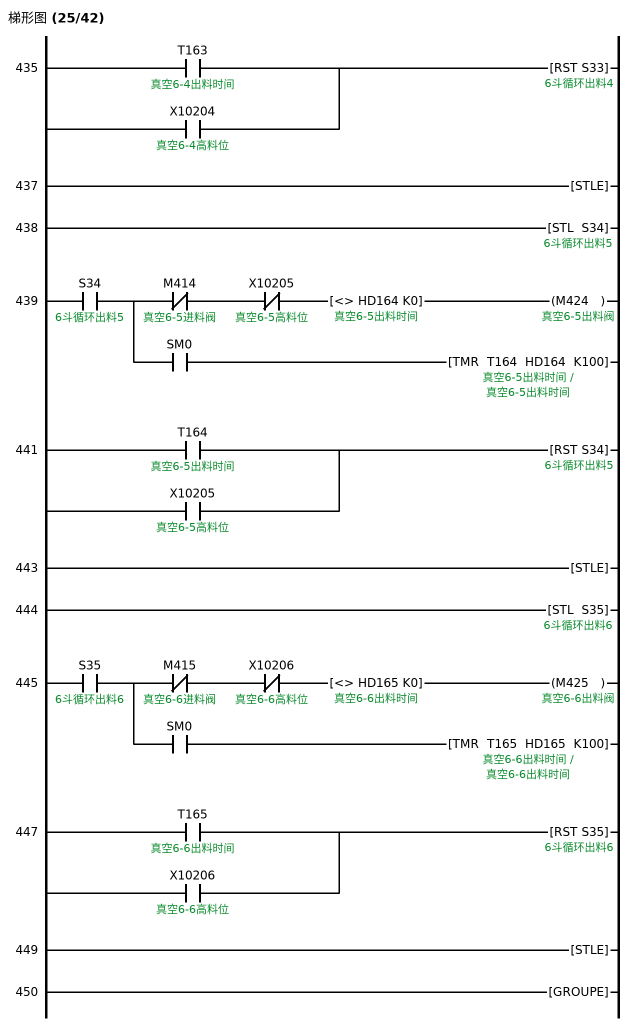
[picture p24: 梯形图 rows 435-450]
LD     T163	; 真空6-4出料时间
OR     X10204	; 真空6-4高料位
RST    S33	; 6斗循环出料4
STLE
STL    S34	; 6斗循环出料5
LD     S34	; 6斗循环出料5
MPS
ANI    M414	; 真空6-5进料阀
ANI    X10205	; 真空6-5高料位
AND<>  HD164 K0	; 真空6-5出料时间
OUT    M424	; 真空6-5出料阀
MPP
AND    SM0
TMR    T164 HD164 K100	; 真空6-5出料时间 / 真空6-5出料时间
LD     T164	; 真空6-5出料时间
OR     X10205	; 真空6-5高料位
RST    S34	; 6斗循环出料5
STLE
STL    S35	; 6斗循环出料6
LD     S35	; 6斗循环出料6
MPS
ANI    M415	; 真空6-6进料阀
ANI    X10206	; 真空6-6高料位
AND<>  HD165 K0	; 真空6-6出料时间
OUT    M425	; 真空6-6出料阀
MPP
AND    SM0
TMR    T165 HD165 K100	; 真空6-6出料时间 / 真空6-6出料时间
LD     T165	; 真空6-6出料时间
OR     X10206	; 真空6-6高料位
RST    S35	; 6斗循环出料6
STLE
GROUPE

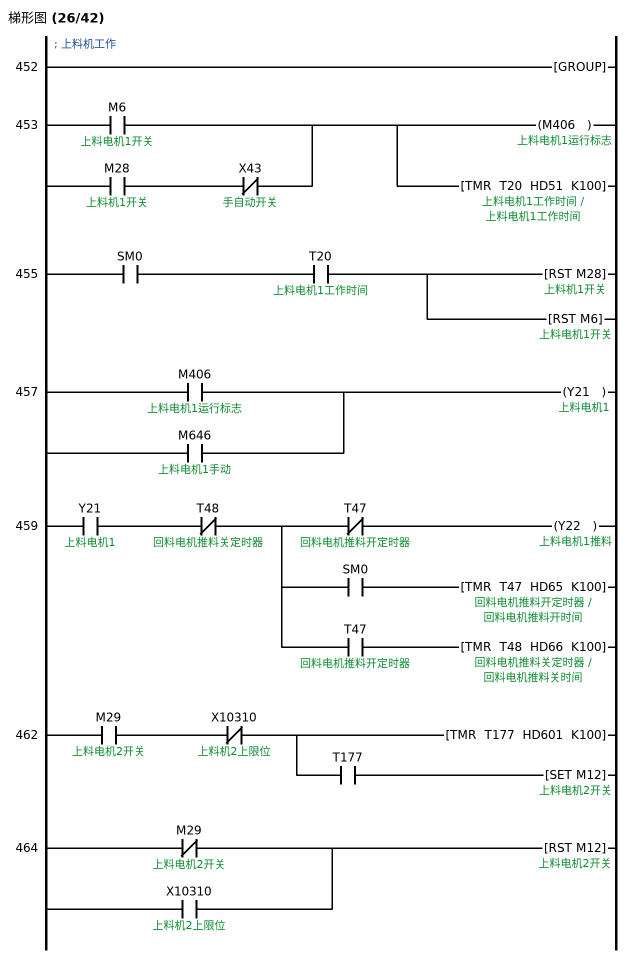
; 上料机工作
GROUP
LD     M6	; 上料电机1开关
LD     M28	; 上料机1开关
ANI    X43	; 手自动开关
ORB
OUT    M406	; 上料电机1运行标志
TMR    T20 HD51 K100	; 上料电机1工作时间 / 上料电机1工作时间
LD     SM0
AND    T20	; 上料电机1工作时间
RST    M28	; 上料机1开关
RST    M6	; 上料电机1开关
LD     M406	; 上料电机1运行标志
OR     M646	; 上料电机1手动
OUT    Y21	; 上料电机1
LD     Y21	; 上料电机1
ANI    T48	; 回料电机推料关定时器
MPS
ANI    T47	; 回料电机推料开定时器
OUT    Y22	; 上料电机1推料
MRD
AND    SM0
TMR    T47 HD65 K100	; 回料电机推料开定时器 / 回料电机推料开时间
MPP
AND    T47	; 回料电机推料开定时器
TMR    T48 HD66 K100	; 回料电机推料关定时器 / 回料电机推料关时间
LD     M29	; 上料电机2开关
ANI    X10310	; 上料机2上限位
TMR    T177 HD601 K100
AND    T177
SET    M12	; 上料电机2开关
LDI    M29	; 上料电机2开关
OR     X10310	; 上料机2上限位
RST    M12	; 上料电机2开关

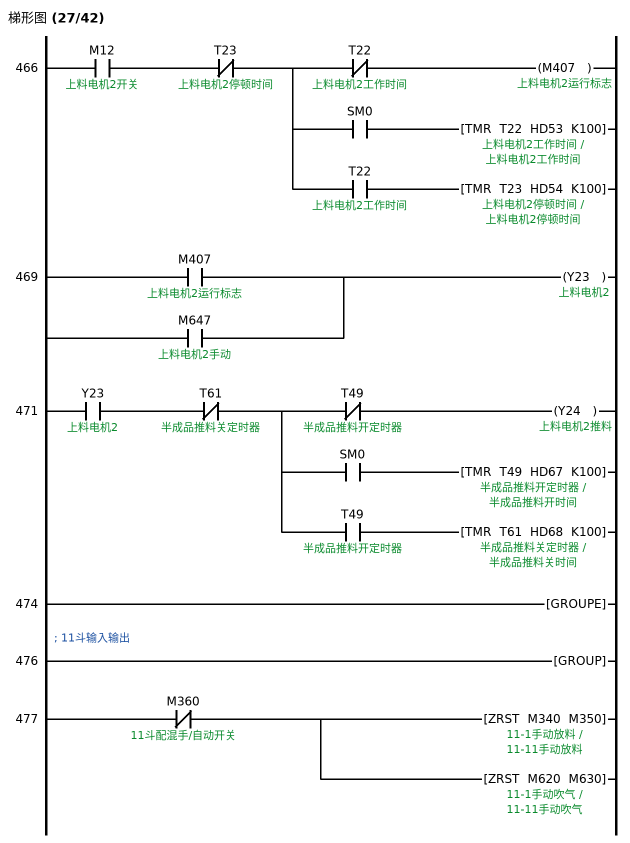
LD     M12	; 上料电机2开关
ANI    T23	; 上料电机2停顿时间
MPS
ANI    T22	; 上料电机2工作时间
OUT    M407	; 上料电机2运行标志
MRD
AND    SM0
TMR    T22 HD53 K100	; 上料电机2工作时间 / 上料电机2工作时间
MPP
AND    T22	; 上料电机2工作时间
TMR    T23 HD54 K100	; 上料电机2停顿时间 / 上料电机2停顿时间
LD     M407	; 上料电机2运行标志
OR     M647	; 上料电机2手动
OUT    Y23	; 上料电机2
LD     Y23	; 上料电机2
ANI    T61	; 半成品推料关定时器
MPS
ANI    T49	; 半成品推料开定时器
OUT    Y24	; 上料电机2推料
MRD
AND    SM0
TMR    T49 HD67 K100	; 半成品推料开定时器 / 半成品推料开时间
MPP
AND    T49	; 半成品推料开定时器
TMR    T61 HD68 K100	; 半成品推料关定时器 / 半成品推料关时间
GROUPE
; 11斗输入输出
GROUP
LDI    M360	; 11斗配混手/自动开关
ZRST   M340 M350	; 11-1手动放料 / 11-11手动放料
ZRST   M620 M630	; 11-1手动吹气 / 11-11手动吹气

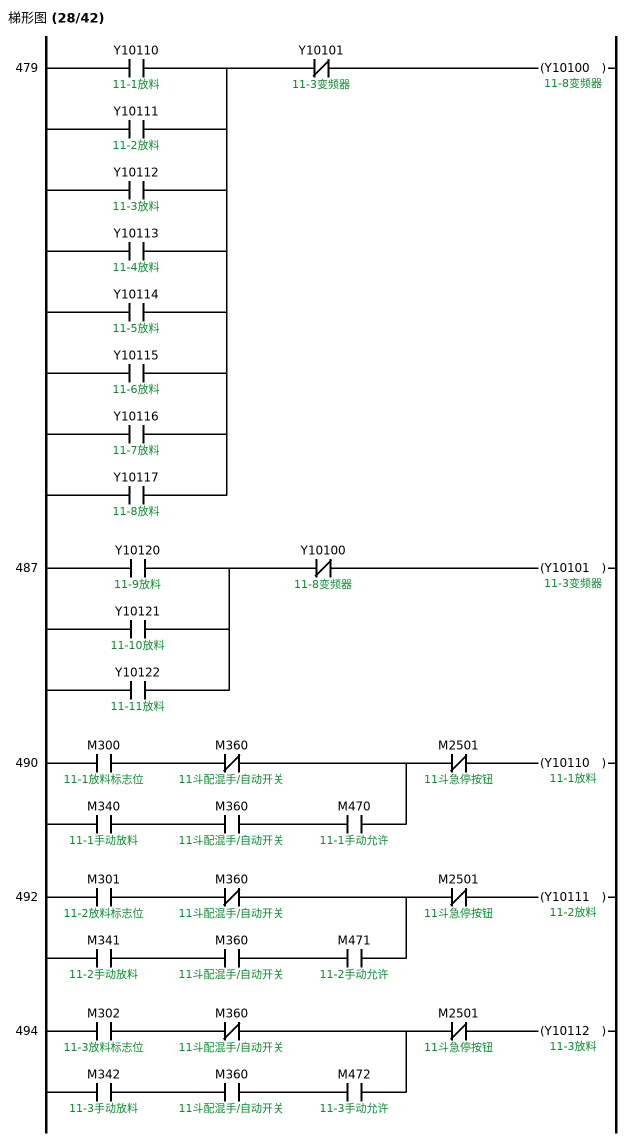
LD     Y10110	; 11-1放料
OR     Y10111	; 11-2放料
OR     Y10112	; 11-3放料
OR     Y10113	; 11-4放料
OR     Y10114	; 11-5放料
OR     Y10115	; 11-6放料
OR     Y10116	; 11-7放料
OR     Y10117	; 11-8放料
ANI    Y10101	; 11-3变频器
OUT    Y10100	; 11-8变频器
LD     Y10120	; 11-9放料
OR     Y10121	; 11-10放料
OR     Y10122	; 11-11放料
ANI    Y10100	; 11-8变频器
OUT    Y10101	; 11-3变频器
LD     M300	; 11-1放料标志位
ANI    M360	; 11斗配混手/自动开关
LD     M340	; 11-1手动放料
AND    M360	; 11斗配混手/自动开关
AND    M470	; 11-1手动允许
ORB
ANI    M2501	; 11斗急停按钮
OUT    Y10110	; 11-1放料
LD     M301	; 11-2放料标志位
ANI    M360	; 11斗配混手/自动开关
LD     M341	; 11-2手动放料
AND    M360	; 11斗配混手/自动开关
AND    M471	; 11-2手动允许
ORB
ANI    M2501	; 11斗急停按钮
OUT    Y10111	; 11-2放料
LD     M302	; 11-3放料标志位
ANI    M360	; 11斗配混手/自动开关
LD     M342	; 11-3手动放料
AND    M360	; 11斗配混手/自动开关
AND    M472	; 11-3手动允许
ORB
ANI    M2501	; 11斗急停按钮
OUT    Y10112	; 11-3放料

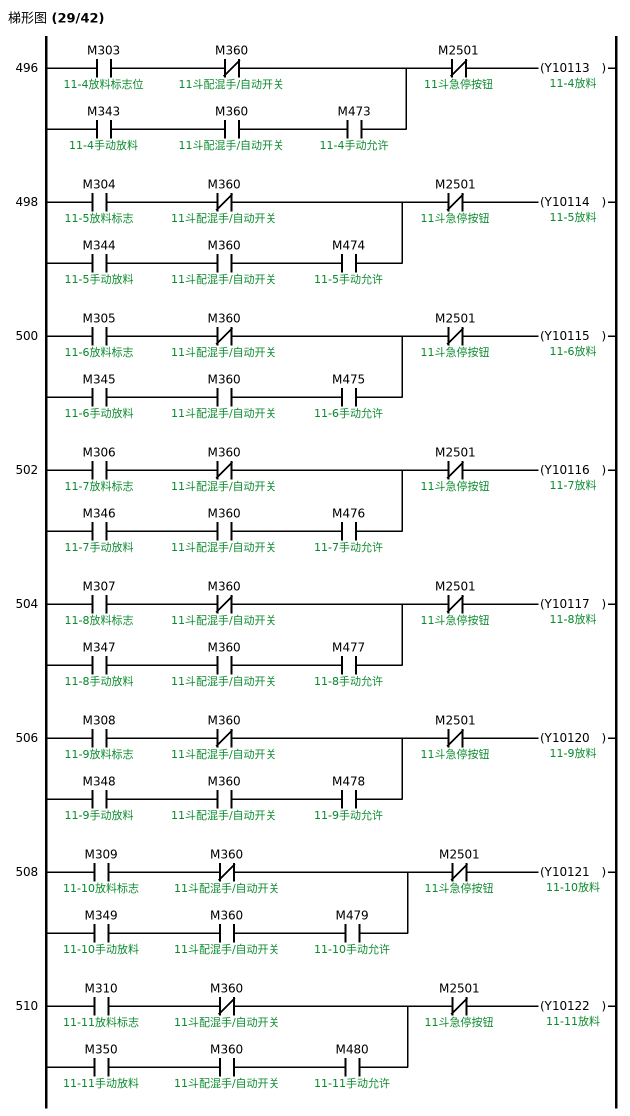
LD     M303	; 11-4放料标志位
ANI    M360	; 11斗配混手/自动开关
LD     M343	; 11-4手动放料
AND    M360	; 11斗配混手/自动开关
AND    M473	; 11-4手动允许
ORB
ANI    M2501	; 11斗急停按钮
OUT    Y10113	; 11-4放料
LD     M304	; 11-5放料标志
ANI    M360	; 11斗配混手/自动开关
LD     M344	; 11-5手动放料
AND    M360	; 11斗配混手/自动开关
AND    M474	; 11-5手动允许
ORB
ANI    M2501	; 11斗急停按钮
OUT    Y10114	; 11-5放料
LD     M305	; 11-6放料标志
ANI    M360	; 11斗配混手/自动开关
LD     M345	; 11-6手动放料
AND    M360	; 11斗配混手/自动开关
AND    M475	; 11-6手动允许
ORB
ANI    M2501	; 11斗急停按钮
OUT    Y10115	; 11-6放料
LD     M306	; 11-7放料标志
ANI    M360	; 11斗配混手/自动开关
LD     M346	; 11-7手动放料
AND    M360	; 11斗配混手/自动开关
AND    M476	; 11-7手动允许
ORB
ANI    M2501	; 11斗急停按钮
OUT    Y10116	; 11-7放料
LD     M307	; 11-8放料标志
ANI    M360	; 11斗配混手/自动开关
LD     M347	; 11-8手动放料
AND    M360	; 11斗配混手/自动开关
AND    M477	; 11-8手动允许
ORB
ANI    M2501	; 11斗急停按钮
OUT    Y10117	; 11-8放料
LD     M308	; 11-9放料标志
ANI    M360	; 11斗配混手/自动开关
LD     M348	; 11-9手动放料
AND    M360	; 11斗配混手/自动开关
AND    M478	; 11-9手动允许
ORB
ANI    M2501	; 11斗急停按钮
OUT    Y10120	; 11-9放料
LD     M309	; 11-10放料标志
ANI    M360	; 11斗配混手/自动开关
LD     M349	; 11-10手动放料
AND    M360	; 11斗配混手/自动开关
AND    M479	; 11-10手动允许
ORB
ANI    M2501	; 11斗急停按钮
OUT    Y10121	; 11-10放料
LD     M310	; 11-11放料标志
ANI    M360	; 11斗配混手/自动开关
LD     M350	; 11-11手动放料
AND    M360	; 11斗配混手/自动开关
AND    M480	; 11-11手动允许
ORB
ANI    M2501	; 11斗急停按钮
OUT    Y10122	; 11-11放料

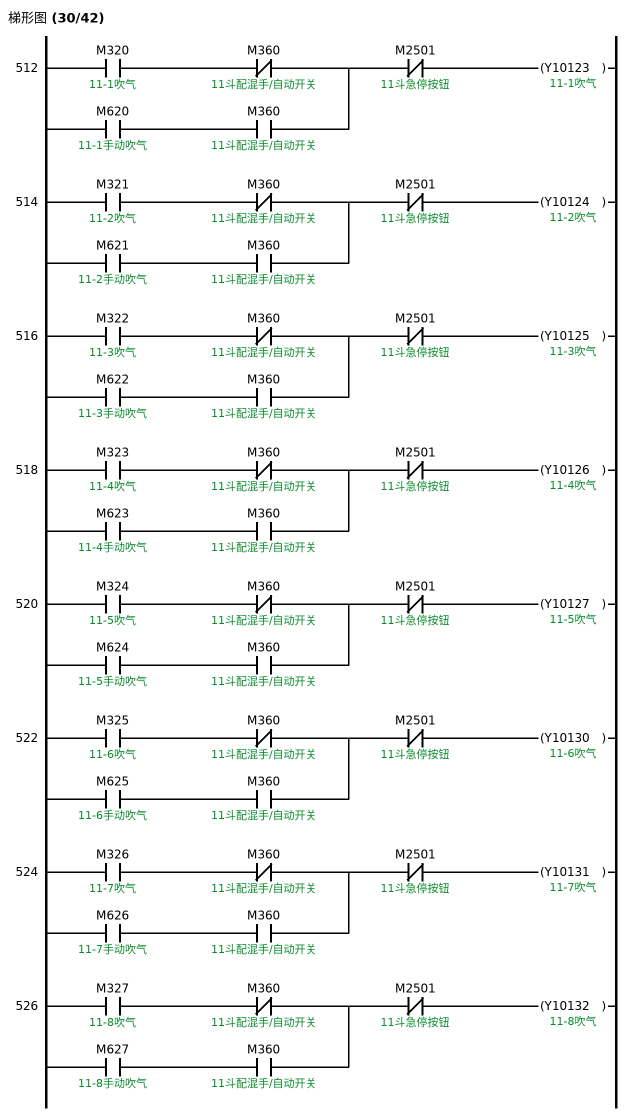
LD     M320	; 11-1吹气
ANI    M360	; 11斗配混手/自动开关
LD     M620	; 11-1手动吹气
AND    M360	; 11斗配混手/自动开关
ORB
ANI    M2501	; 11斗急停按钮
OUT    Y10123	; 11-1吹气
LD     M321	; 11-2吹气
ANI    M360	; 11斗配混手/自动开关
LD     M621	; 11-2手动吹气
AND    M360	; 11斗配混手/自动开关
ORB
ANI    M2501	; 11斗急停按钮
OUT    Y10124	; 11-2吹气
LD     M322	; 11-3吹气
ANI    M360	; 11斗配混手/自动开关
LD     M622	; 11-3手动吹气
AND    M360	; 11斗配混手/自动开关
ORB
ANI    M2501	; 11斗急停按钮
OUT    Y10125	; 11-3吹气
LD     M323	; 11-4吹气
ANI    M360	; 11斗配混手/自动开关
LD     M623	; 11-4手动吹气
AND    M360	; 11斗配混手/自动开关
ORB
ANI    M2501	; 11斗急停按钮
OUT    Y10126	; 11-4吹气
LD     M324	; 11-5吹气
ANI    M360	; 11斗配混手/自动开关
LD     M624	; 11-5手动吹气
AND    M360	; 11斗配混手/自动开关
ORB
ANI    M2501	; 11斗急停按钮
OUT    Y10127	; 11-5吹气
LD     M325	; 11-6吹气
ANI    M360	; 11斗配混手/自动开关
LD     M625	; 11-6手动吹气
AND    M360	; 11斗配混手/自动开关
ORB
ANI    M2501	; 11斗急停按钮
OUT    Y10130	; 11-6吹气
LD     M326	; 11-7吹气
ANI    M360	; 11斗配混手/自动开关
LD     M626	; 11-7手动吹气
AND    M360	; 11斗配混手/自动开关
ORB
ANI    M2501	; 11斗急停按钮
OUT    Y10131	; 11-7吹气
LD     M327	; 11-8吹气
ANI    M360	; 11斗配混手/自动开关
LD     M627	; 11-8手动吹气
AND    M360	; 11斗配混手/自动开关
ORB
ANI    M2501	; 11斗急停按钮
OUT    Y10132	; 11-8吹气

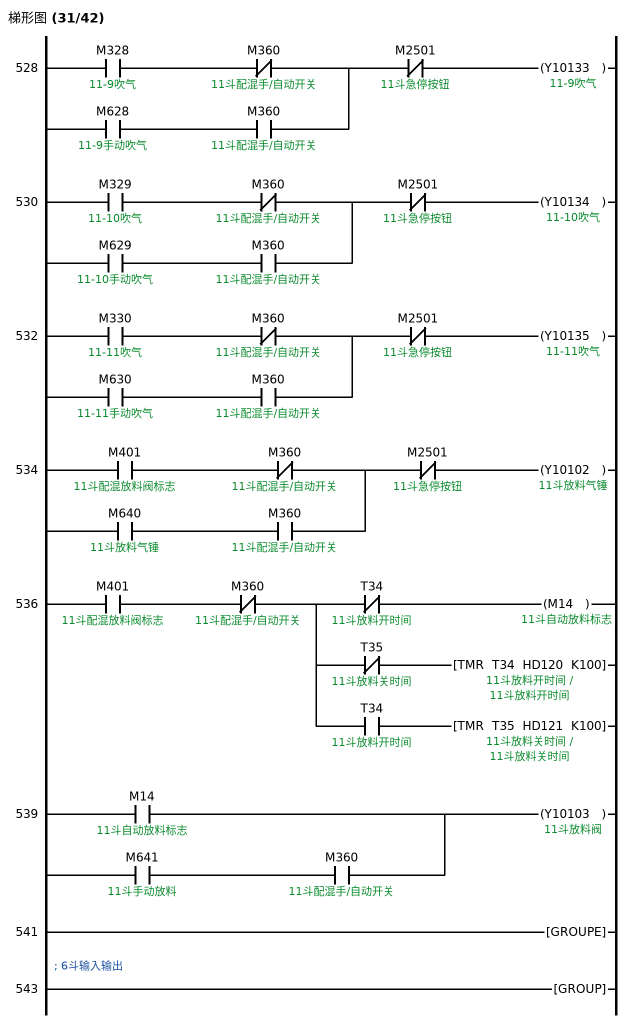
LD     M328	; 11-9吹气
ANI    M360	; 11斗配混手/自动开关
LD     M628	; 11-9手动吹气
AND    M360	; 11斗配混手/自动开关
ORB
ANI    M2501	; 11斗急停按钮
OUT    Y10133	; 11-9吹气
LD     M329	; 11-10吹气
ANI    M360	; 11斗配混手/自动开关
LD     M629	; 11-10手动吹气
AND    M360	; 11斗配混手/自动开关
ORB
ANI    M2501	; 11斗急停按钮
OUT    Y10134	; 11-10吹气
LD     M330	; 11-11吹气
ANI    M360	; 11斗配混手/自动开关
LD     M630	; 11-11手动吹气
AND    M360	; 11斗配混手/自动开关
ORB
ANI    M2501	; 11斗急停按钮
OUT    Y10135	; 11-11吹气
LD     M401	; 11斗配混放料阀标志
ANI    M360	; 11斗配混手/自动开关
LD     M640	; 11斗放料气锤
AND    M360	; 11斗配混手/自动开关
ORB
ANI    M2501	; 11斗急停按钮
OUT    Y10102	; 11斗放料气锤
LD     M401	; 11斗配混放料阀标志
ANI    M360	; 11斗配混手/自动开关
MPS
ANI    T34	; 11斗放料开时间
OUT    M14	; 11斗自动放料标志
MRD
ANI    T35	; 11斗放料关时间
TMR    T34 HD120 K100	; 11斗放料开时间 / 11斗放料开时间
MPP
AND    T34	; 11斗放料开时间
TMR    T35 HD121 K100	; 11斗放料关时间 / 11斗放料关时间
LD     M14	; 11斗自动放料标志
LD     M641	; 11斗手动放料
AND    M360	; 11斗配混手/自动开关
ORB
OUT    Y10103	; 11斗放料阀
GROUPE
; 6斗输入输出
GROUP

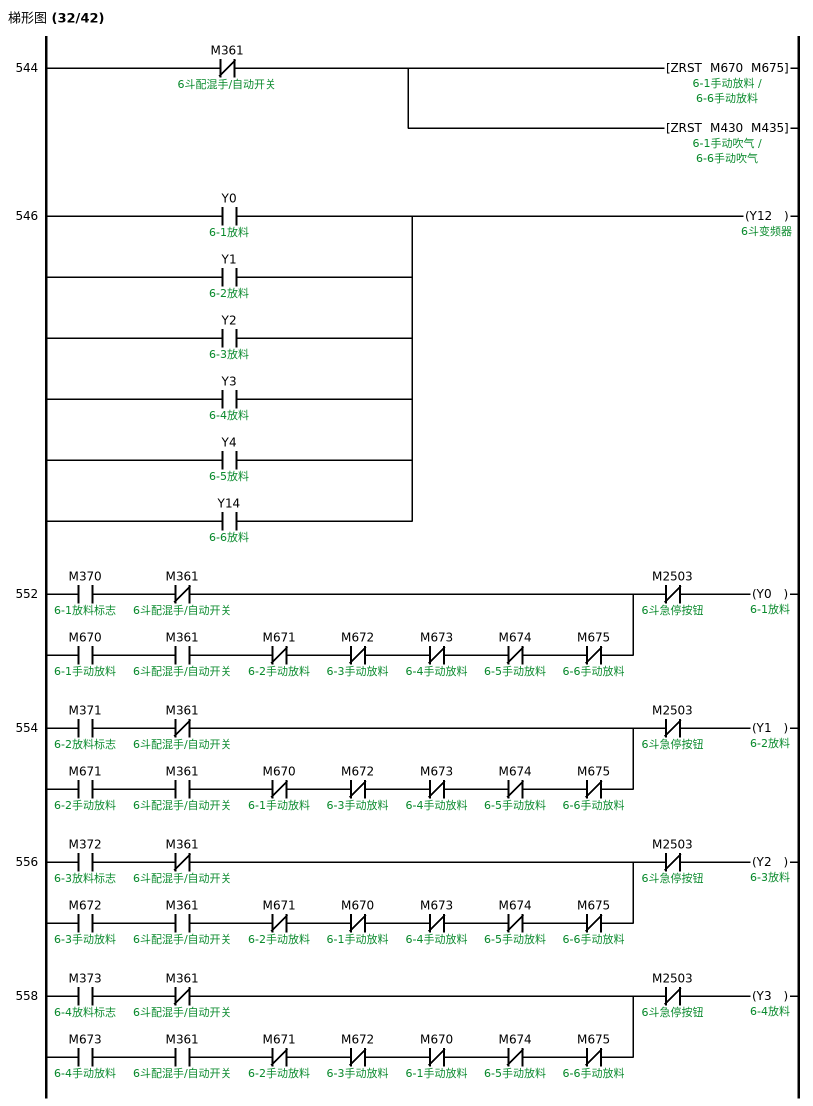
LDI    M361	; 6斗配混手/自动开关
ZRST   M670 M675	; 6-1手动放料 / 6-6手动放料
ZRST   M430 M435	; 6-1手动吹气 / 6-6手动吹气
LD     Y0	; 6-1放料
OR     Y1	; 6-2放料
OR     Y2	; 6-3放料
OR     Y3	; 6-4放料
OR     Y4	; 6-5放料
OR     Y14	; 6-6放料
OUT    Y12	; 6斗变频器
LD     M370	; 6-1放料标志
ANI    M361	; 6斗配混手/自动开关
LD     M670	; 6-1手动放料
AND    M361	; 6斗配混手/自动开关
ANI    M671	; 6-2手动放料
ANI    M672	; 6-3手动放料
ANI    M673	; 6-4手动放料
ANI    M674	; 6-5手动放料
ANI    M675	; 6-6手动放料
ORB
ANI    M2503	; 6斗急停按钮
OUT    Y0	; 6-1放料
LD     M371	; 6-2放料标志
ANI    M361	; 6斗配混手/自动开关
LD     M671	; 6-2手动放料
AND    M361	; 6斗配混手/自动开关
ANI    M670	; 6-1手动放料
ANI    M672	; 6-3手动放料
ANI    M673	; 6-4手动放料
ANI    M674	; 6-5手动放料
ANI    M675	; 6-6手动放料
ORB
ANI    M2503	; 6斗急停按钮
OUT    Y1	; 6-2放料
LD     M372	; 6-3放料标志
ANI    M361	; 6斗配混手/自动开关
LD     M672	; 6-3手动放料
AND    M361	; 6斗配混手/自动开关
ANI    M671	; 6-2手动放料
ANI    M670	; 6-1手动放料
ANI    M673	; 6-4手动放料
ANI    M674	; 6-5手动放料
ANI    M675	; 6-6手动放料
ORB
ANI    M2503	; 6斗急停按钮
OUT    Y2	; 6-3放料
LD     M373	; 6-4放料标志
ANI    M361	; 6斗配混手/自动开关
LD     M673	; 6-4手动放料
AND    M361	; 6斗配混手/自动开关
ANI    M671	; 6-2手动放料
ANI    M672	; 6-3手动放料
ANI    M670	; 6-1手动放料
ANI    M674	; 6-5手动放料
ANI    M675	; 6-6手动放料
ORB
ANI    M2503	; 6斗急停按钮
OUT    Y3	; 6-4放料

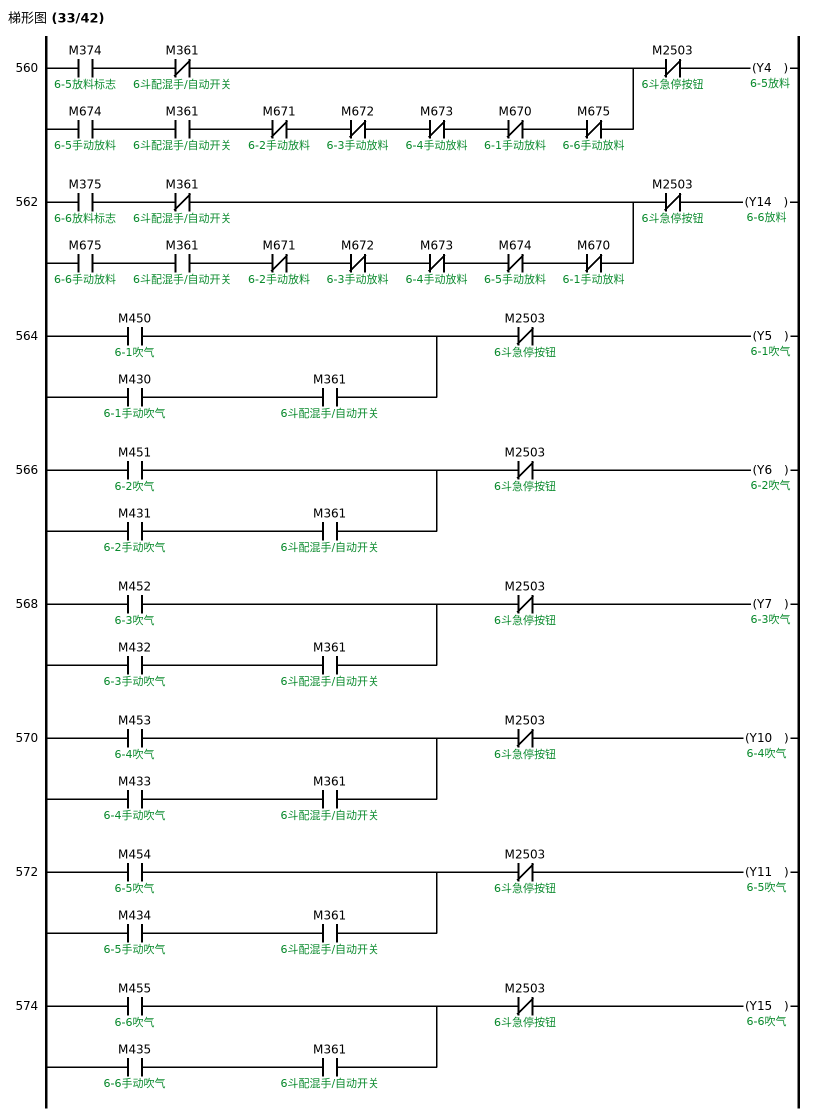
LD     M374	; 6-5放料标志
ANI    M361	; 6斗配混手/自动开关
LD     M674	; 6-5手动放料
AND    M361	; 6斗配混手/自动开关
ANI    M671	; 6-2手动放料
ANI    M672	; 6-3手动放料
ANI    M673	; 6-4手动放料
ANI    M670	; 6-1手动放料
ANI    M675	; 6-6手动放料
ORB
ANI    M2503	; 6斗急停按钮
OUT    Y4	; 6-5放料
LD     M375	; 6-6放料标志
ANI    M361	; 6斗配混手/自动开关
LD     M675	; 6-6手动放料
AND    M361	; 6斗配混手/自动开关
ANI    M671	; 6-2手动放料
ANI    M672	; 6-3手动放料
ANI    M673	; 6-4手动放料
ANI    M674	; 6-5手动放料
ANI    M670	; 6-1手动放料
ORB
ANI    M2503	; 6斗急停按钮
OUT    Y14	; 6-6放料
LD     M450	; 6-1吹气
LD     M430	; 6-1手动吹气
AND    M361	; 6斗配混手/自动开关
ORB
ANI    M2503	; 6斗急停按钮
OUT    Y5	; 6-1吹气
LD     M451	; 6-2吹气
LD     M431	; 6-2手动吹气
AND    M361	; 6斗配混手/自动开关
ORB
ANI    M2503	; 6斗急停按钮
OUT    Y6	; 6-2吹气
LD     M452	; 6-3吹气
LD     M432	; 6-3手动吹气
AND    M361	; 6斗配混手/自动开关
ORB
ANI    M2503	; 6斗急停按钮
OUT    Y7	; 6-3吹气
LD     M453	; 6-4吹气
LD     M433	; 6-4手动吹气
AND    M361	; 6斗配混手/自动开关
ORB
ANI    M2503	; 6斗急停按钮
OUT    Y10	; 6-4吹气
LD     M454	; 6-5吹气
LD     M434	; 6-5手动吹气
AND    M361	; 6斗配混手/自动开关
ORB
ANI    M2503	; 6斗急停按钮
OUT    Y11	; 6-5吹气
LD     M455	; 6-6吹气
LD     M435	; 6-6手动吹气
AND    M361	; 6斗配混手/自动开关
ORB
ANI    M2503	; 6斗急停按钮
OUT    Y15	; 6-6吹气

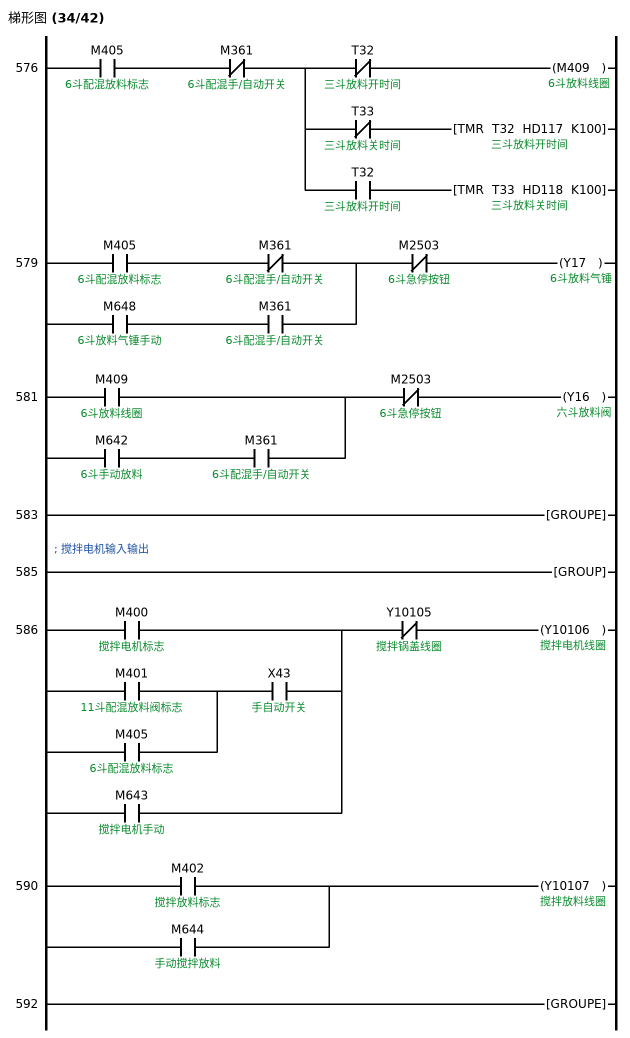
LD     M405	; 6斗配混放料标志
ANI    M361	; 6斗配混手/自动开关
MPS
ANI    T32	; 三斗放料开时间
OUT    M409	; 6斗放料线圈
MRD
ANI    T33	; 三斗放料关时间
TMR    T32 HD117 K100	; 三斗放料开时间
MPP
AND    T32	; 三斗放料开时间
TMR    T33 HD118 K100	; 三斗放料关时间
LD     M405	; 6斗配混放料标志
ANI    M361	; 6斗配混手/自动开关
LD     M648	; 6斗放料气锤手动
AND    M361	; 6斗配混手/自动开关
ORB
ANI    M2503	; 6斗急停按钮
OUT    Y17	; 6斗放料气锤
LD     M409	; 6斗放料线圈
LD     M642	; 6斗手动放料
AND    M361	; 6斗配混手/自动开关
ORB
ANI    M2503	; 6斗急停按钮
OUT    Y16	; 六斗放料阀
GROUPE
; 搅拌电机输入输出
GROUP
LD     M400	; 搅拌电机标志
LD     M401	; 11斗配混放料阀标志
OR     M405	; 6斗配混放料标志
AND    X43	; 手自动开关
ORB
OR     M643	; 搅拌电机手动
ANI    Y10105	; 搅拌锅盖线圈
OUT    Y10106	; 搅拌电机线圈
LD     M402	; 搅拌放料标志
OR     M644	; 手动搅拌放料
OUT    Y10107	; 搅拌放料线圈
GROUPE

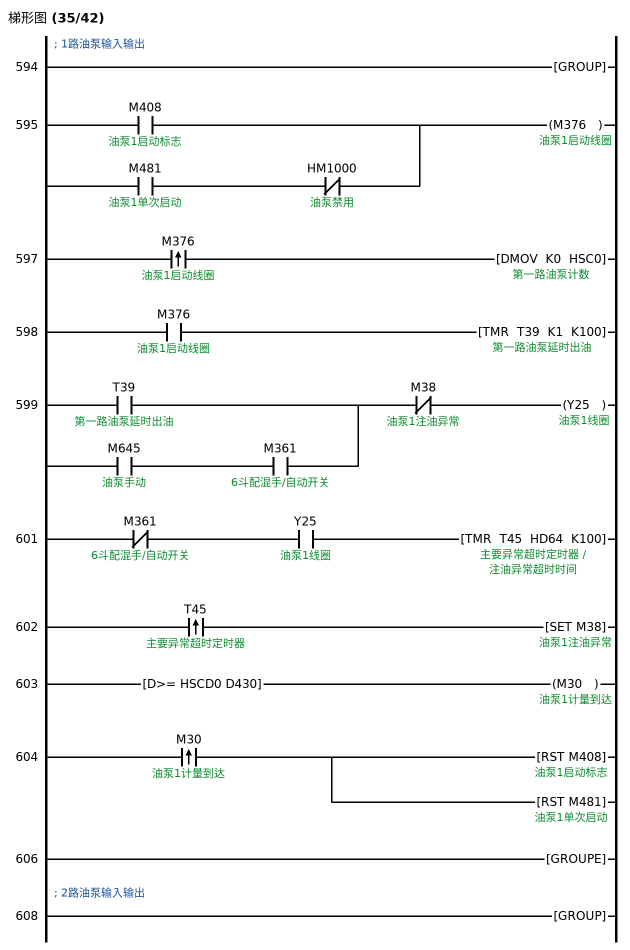
; 1路油泵输入输出
GROUP
LD     M408	; 油泵1启动标志
LD     M481	; 油泵1单次启动
ANI    HM1000	; 油泵禁用
ORB
OUT    M376	; 油泵1启动线圈
LDP    M376	; 油泵1启动线圈
DMOV   K0 HSC0	; 第一路油泵计数
LD     M376	; 油泵1启动线圈
TMR    T39 K1 K100	; 第一路油泵延时出油
LD     T39	; 第一路油泵延时出油
LD     M645	; 油泵手动
AND    M361	; 6斗配混手/自动开关
ORB
ANI    M38	; 油泵1注油异常
OUT    Y25	; 油泵1线圈
LDI    M361	; 6斗配混手/自动开关
AND    Y25	; 油泵1线圈
TMR    T45 HD64 K100	; 主要异常超时定时器 / 注油异常超时时间
LDP    T45	; 主要异常超时定时器
SET    M38	; 油泵1注油异常
DLD>=  HSCD0 D430
OUT    M30	; 油泵1计量到达
LDP    M30	; 油泵1计量到达
RST    M408	; 油泵1启动标志
RST    M481	; 油泵1单次启动
GROUPE
; 2路油泵输入输出
GROUP

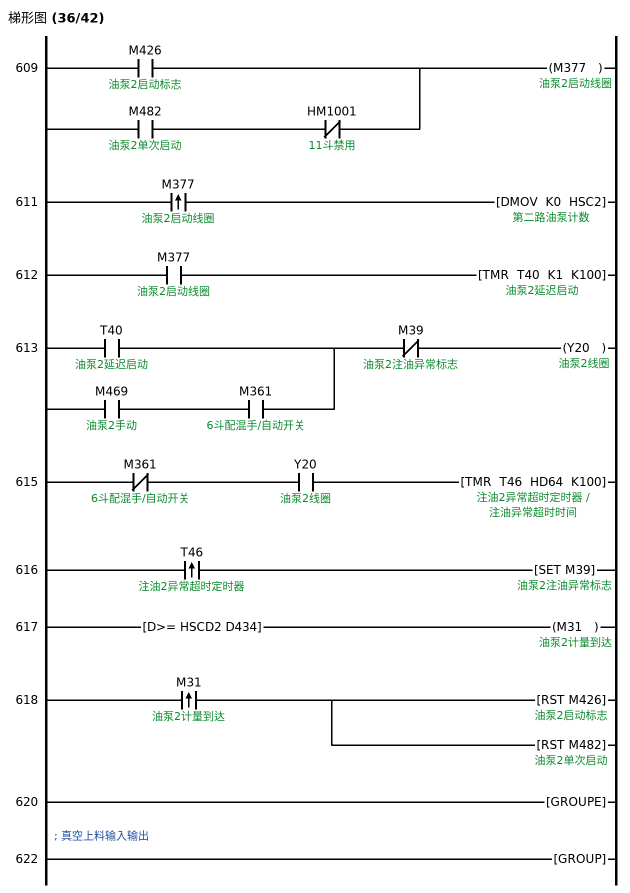
LD     M426	; 油泵2启动标志
LD     M482	; 油泵2单次启动
ANI    HM1001	; 11斗禁用
ORB
OUT    M377	; 油泵2启动线圈
LDP    M377	; 油泵2启动线圈
DMOV   K0 HSC2	; 第二路油泵计数
LD     M377	; 油泵2启动线圈
TMR    T40 K1 K100	; 油泵2延迟启动
LD     T40	; 油泵2延迟启动
LD     M469	; 油泵2手动
AND    M361	; 6斗配混手/自动开关
ORB
ANI    M39	; 油泵2注油异常标志
OUT    Y20	; 油泵2线圈
LDI    M361	; 6斗配混手/自动开关
AND    Y20	; 油泵2线圈
TMR    T46 HD64 K100	; 注油2异常超时定时器 / 注油异常超时时间
LDP    T46	; 注油2异常超时定时器
SET    M39	; 油泵2注油异常标志
DLD>=  HSCD2 D434
OUT    M31	; 油泵2计量到达
LDP    M31	; 油泵2计量到达
RST    M426	; 油泵2启动标志
RST    M482	; 油泵2单次启动
GROUPE
; 真空上料输入输出
GROUP

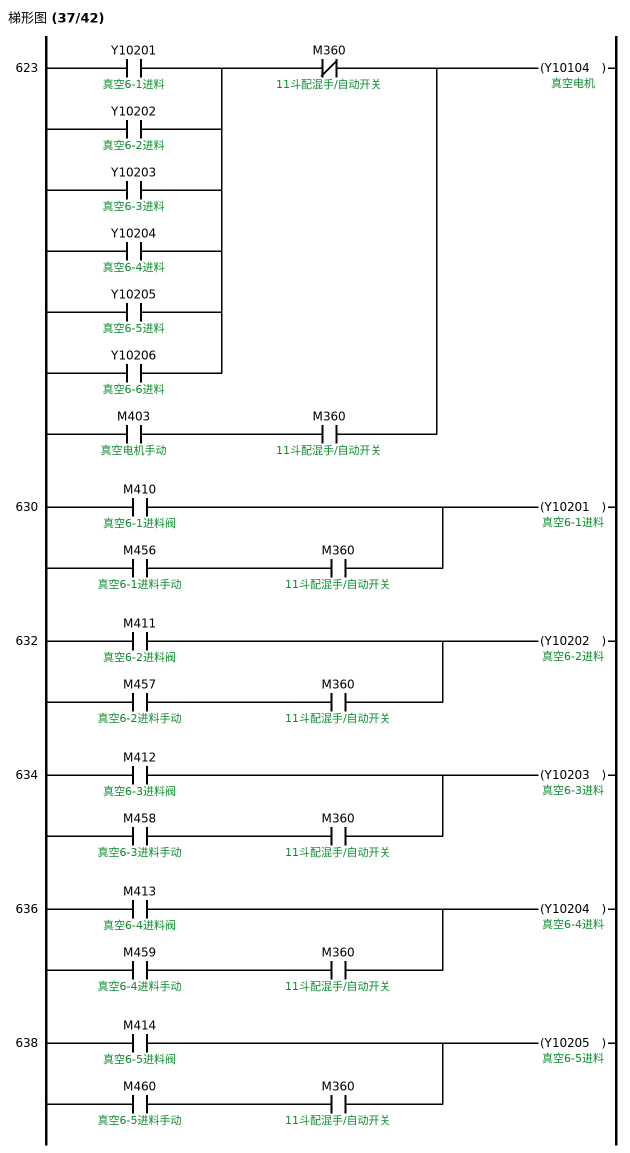
LD     Y10201	; 真空6-1进料
OR     Y10202	; 真空6-2进料
OR     Y10203	; 真空6-3进料
OR     Y10204	; 真空6-4进料
OR     Y10205	; 真空6-5进料
OR     Y10206	; 真空6-6进料
ANI    M360	; 11斗配混手/自动开关
LD     M403	; 真空电机手动
AND    M360	; 11斗配混手/自动开关
ORB
OUT    Y10104	; 真空电机
LD     M410	; 真空6-1进料阀
LD     M456	; 真空6-1进料手动
AND    M360	; 11斗配混手/自动开关
ORB
OUT    Y10201	; 真空6-1进料
LD     M411	; 真空6-2进料阀
LD     M457	; 真空6-2进料手动
AND    M360	; 11斗配混手/自动开关
ORB
OUT    Y10202	; 真空6-2进料
LD     M412	; 真空6-3进料阀
LD     M458	; 真空6-3进料手动
AND    M360	; 11斗配混手/自动开关
ORB
OUT    Y10203	; 真空6-3进料
LD     M413	; 真空6-4进料阀
LD     M459	; 真空6-4进料手动
AND    M360	; 11斗配混手/自动开关
ORB
OUT    Y10204	; 真空6-4进料
LD     M414	; 真空6-5进料阀
LD     M460	; 真空6-5进料手动
AND    M360	; 11斗配混手/自动开关
ORB
OUT    Y10205	; 真空6-5进料

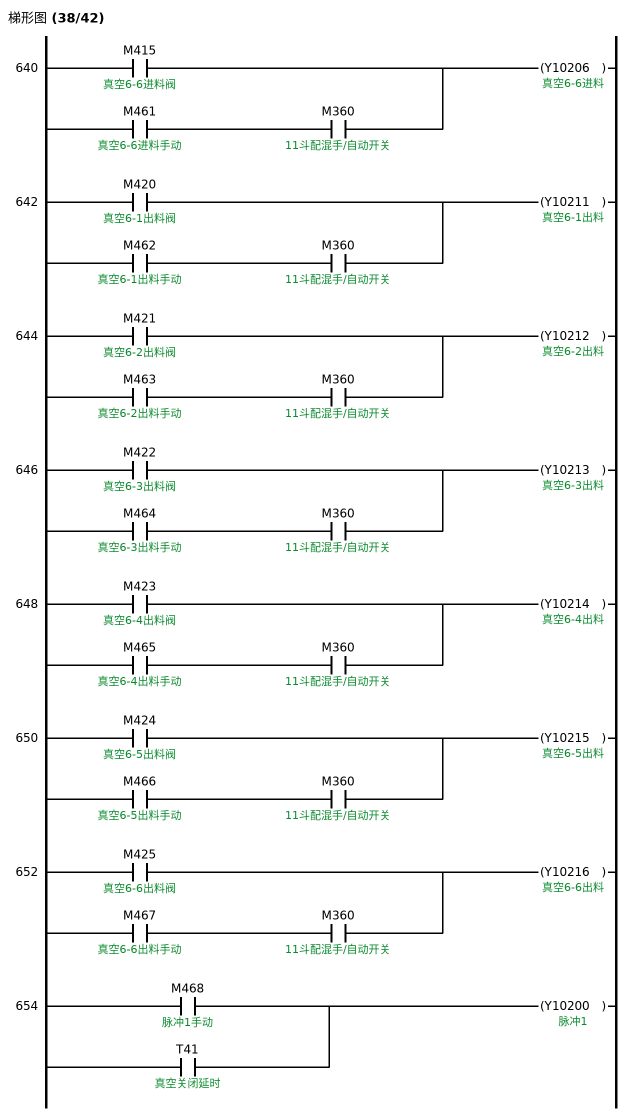
LD     M415	; 真空6-6进料阀
LD     M461	; 真空6-6进料手动
AND    M360	; 11斗配混手/自动开关
ORB
OUT    Y10206	; 真空6-6进料
LD     M420	; 真空6-1出料阀
LD     M462	; 真空6-1出料手动
AND    M360	; 11斗配混手/自动开关
ORB
OUT    Y10211	; 真空6-1出料
LD     M421	; 真空6-2出料阀
LD     M463	; 真空6-2出料手动
AND    M360	; 11斗配混手/自动开关
ORB
OUT    Y10212	; 真空6-2出料
LD     M422	; 真空6-3出料阀
LD     M464	; 真空6-3出料手动
AND    M360	; 11斗配混手/自动开关
ORB
OUT    Y10213	; 真空6-3出料
LD     M423	; 真空6-4出料阀
LD     M465	; 真空6-4出料手动
AND    M360	; 11斗配混手/自动开关
ORB
OUT    Y10214	; 真空6-4出料
LD     M424	; 真空6-5出料阀
LD     M466	; 真空6-5出料手动
AND    M360	; 11斗配混手/自动开关
ORB
OUT    Y10215	; 真空6-5出料
LD     M425	; 真空6-6出料阀
LD     M467	; 真空6-6出料手动
AND    M360	; 11斗配混手/自动开关
ORB
OUT    Y10216	; 真空6-6出料
LD     M468	; 脉冲1手动
OR     T41	; 真空关闭延时
OUT    Y10200	; 脉冲1

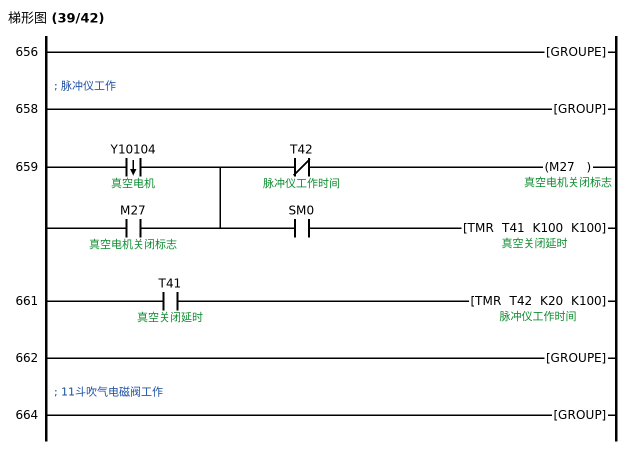
GROUPE
; 脉冲仪工作
GROUP
LDF    Y10104	; 真空电机
OR     M27	; 真空电机关闭标志
MPS
ANI    T42	; 脉冲仪工作时间
OUT    M27	; 真空电机关闭标志
MPP
AND    SM0
TMR    T41 K100 K100	; 真空关闭延时
LD     T41	; 真空关闭延时
TMR    T42 K20 K100	; 脉冲仪工作时间
GROUPE
; 11斗吹气电磁阀工作
GROUP

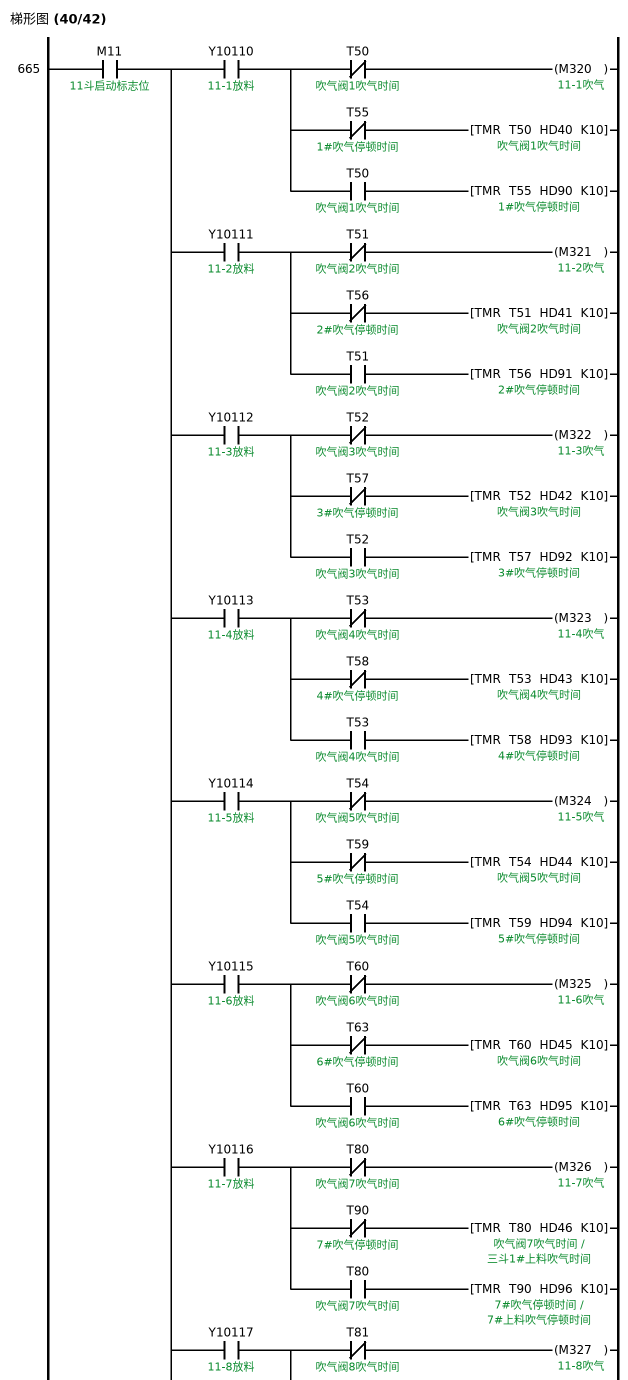
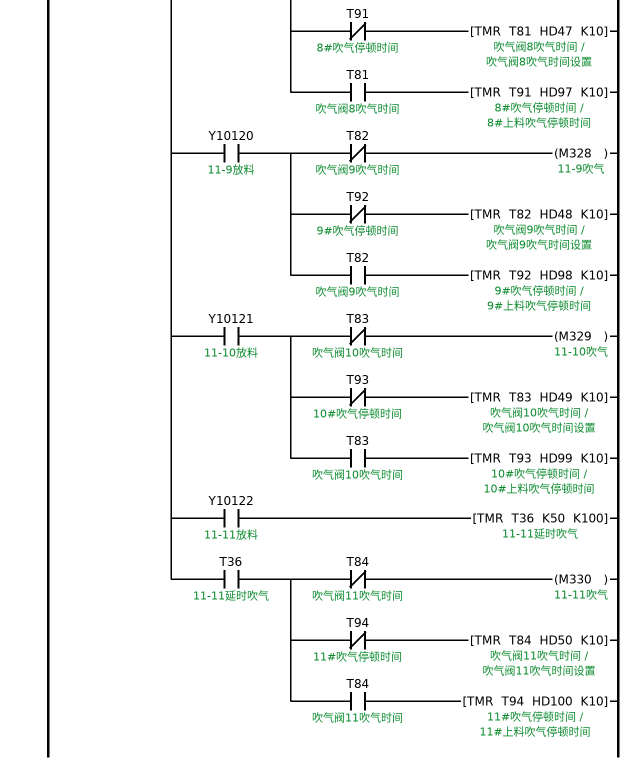
LD     M11	; 11斗启动标志位
MPS
AND    Y10110	; 11-1放料
MPS
ANI    T50	; 吹气阀1吹气时间
OUT    M320	; 11-1吹气
MRD
ANI    T55	; 1#吹气停顿时间
TMR    T50 HD40 K10	; 吹气阀1吹气时间
MPP
AND    T50	; 吹气阀1吹气时间
TMR    T55 HD90 K10	; 1#吹气停顿时间
MRD
AND    Y10111	; 11-2放料
MPS
ANI    T51	; 吹气阀2吹气时间
OUT    M321	; 11-2吹气
MRD
ANI    T56	; 2#吹气停顿时间
TMR    T51 HD41 K10	; 吹气阀2吹气时间
MPP
AND    T51	; 吹气阀2吹气时间
TMR    T56 HD91 K10	; 2#吹气停顿时间
MRD
AND    Y10112	; 11-3放料
MPS
ANI    T52	; 吹气阀3吹气时间
OUT    M322	; 11-3吹气
MRD
ANI    T57	; 3#吹气停顿时间
TMR    T52 HD42 K10	; 吹气阀3吹气时间
MPP
AND    T52	; 吹气阀3吹气时间
TMR    T57 HD92 K10	; 3#吹气停顿时间
MRD
AND    Y10113	; 11-4放料
MPS
ANI    T53	; 吹气阀4吹气时间
OUT    M323	; 11-4吹气
MRD
ANI    T58	; 4#吹气停顿时间
TMR    T53 HD43 K10	; 吹气阀4吹气时间
MPP
AND    T53	; 吹气阀4吹气时间
TMR    T58 HD93 K10	; 4#吹气停顿时间
MRD
AND    Y10114	; 11-5放料
MPS
ANI    T54	; 吹气阀5吹气时间
OUT    M324	; 11-5吹气
MRD
ANI    T59	; 5#吹气停顿时间
TMR    T54 HD44 K10	; 吹气阀5吹气时间
MPP
AND    T54	; 吹气阀5吹气时间
TMR    T59 HD94 K10	; 5#吹气停顿时间
MRD
AND    Y10115	; 11-6放料
MPS
ANI    T60	; 吹气阀6吹气时间
OUT    M325	; 11-6吹气
MRD
ANI    T63	; 6#吹气停顿时间
TMR    T60 HD45 K10	; 吹气阀6吹气时间
MPP
AND    T60	; 吹气阀6吹气时间
TMR    T63 HD95 K10	; 6#吹气停顿时间
MRD
AND    Y10116	; 11-7放料
MPS
ANI    T80	; 吹气阀7吹气时间
OUT    M326	; 11-7吹气
MRD
ANI    T90	; 7#吹气停顿时间
TMR    T80 HD46 K10	; 吹气阀7吹气时间 / 三斗1#上料吹气时间
MPP
AND    T80	; 吹气阀7吹气时间
TMR    T90 HD96 K10	; 7#吹气停顿时间 / 7#上料吹气停顿时间
MRD
AND    Y10117	; 11-8放料
MPS
ANI    T81	; 吹气阀8吹气时间
OUT    M327	; 11-8吹气
MRD
ANI    T91	; 8#吹气停顿时间
TMR    T81 HD47 K10	; 吹气阀8吹气时间 / 吹气阀8吹气时间设置
MPP
AND    T81	; 吹气阀8吹气时间
TMR    T91 HD97 K10	; 8#吹气停顿时间 / 8#上料吹气停顿时间
MRD
AND    Y10120	; 11-9放料
MPS
ANI    T82	; 吹气阀9吹气时间
OUT    M328	; 11-9吹气
MRD
ANI    T92	; 9#吹气停顿时间
TMR    T82 HD48 K10	; 吹气阀9吹气时间 / 吹气阀9吹气时间设置
MPP
AND    T82	; 吹气阀9吹气时间
TMR    T92 HD98 K10	; 9#吹气停顿时间 / 9#上料吹气停顿时间
MRD
AND    Y10121	; 11-10放料
MPS
ANI    T83	; 吹气阀10吹气时间
OUT    M329	; 11-10吹气
MRD
ANI    T93	; 10#吹气停顿时间
TMR    T83 HD49 K10	; 吹气阀10吹气时间 / 吹气阀10吹气时间设置
MPP
AND    T83	; 吹气阀10吹气时间
TMR    T93 HD99 K10	; 10#吹气停顿时间 / 10#上料吹气停顿时间
MRD
AND    Y10122	; 11-11放料
TMR    T36 K50 K100	; 11-11延时吹气
MPP
AND    T36	; 11-11延时吹气
MPS
ANI    T84	; 吹气阀11吹气时间
OUT    M330	; 11-11吹气
MRD
ANI    T94	; 11#吹气停顿时间
TMR    T84 HD50 K10	; 吹气阀11吹气时间 / 吹气阀11吹气时间设置
MPP
AND    T84	; 吹气阀11吹气时间
TMR    T94 HD100 K10	; 11#吹气停顿时间 / 11#上料吹气停顿时间

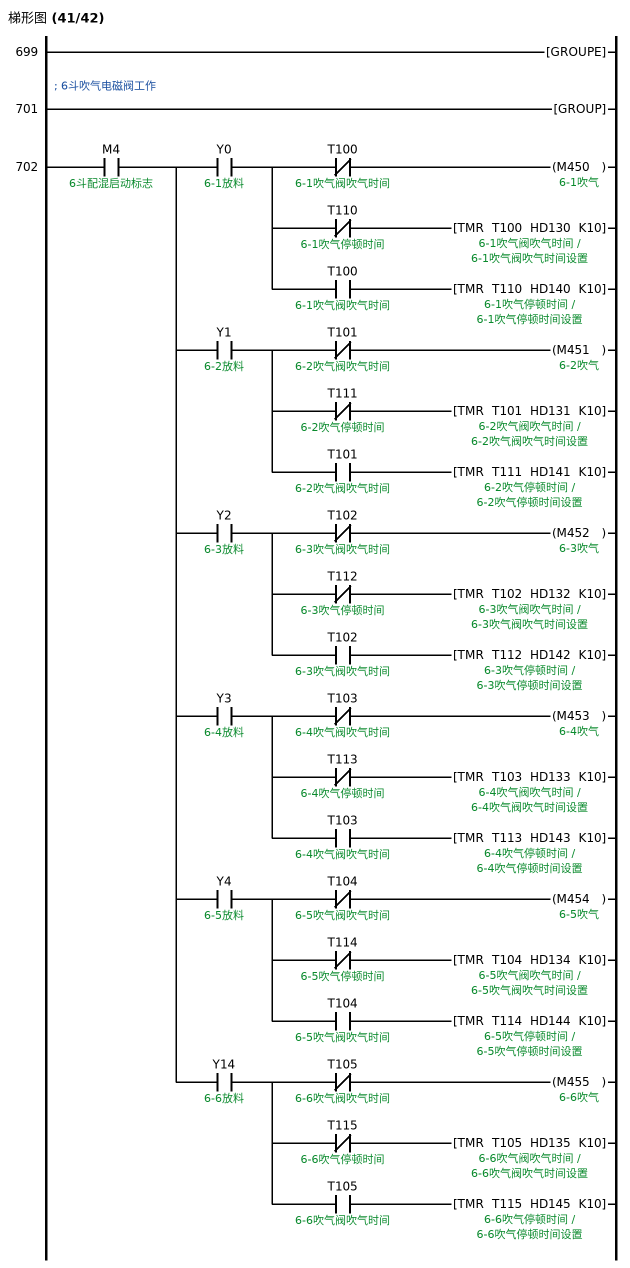
GROUPE
; 6斗吹气电磁阀工作
GROUP
LD     M4	; 6斗配混启动标志
MPS
AND    Y0	; 6-1放料
MPS
ANI    T100	; 6-1吹气阀吹气时间
OUT    M450	; 6-1吹气
MRD
ANI    T110	; 6-1吹气停顿时间
TMR    T100 HD130 K10	; 6-1吹气阀吹气时间 / 6-1吹气阀吹气时间设置
MPP
AND    T100	; 6-1吹气阀吹气时间
TMR    T110 HD140 K10	; 6-1吹气停顿时间 / 6-1吹气停顿时间设置
MRD
AND    Y1	; 6-2放料
MPS
ANI    T101	; 6-2吹气阀吹气时间
OUT    M451	; 6-2吹气
MRD
ANI    T111	; 6-2吹气停顿时间
TMR    T101 HD131 K10	; 6-2吹气阀吹气时间 / 6-2吹气阀吹气时间设置
MPP
AND    T101	; 6-2吹气阀吹气时间
TMR    T111 HD141 K10	; 6-2吹气停顿时间 / 6-2吹气停顿时间设置
MRD
AND    Y2	; 6-3放料
MPS
ANI    T102	; 6-3吹气阀吹气时间
OUT    M452	; 6-3吹气
MRD
ANI    T112	; 6-3吹气停顿时间
TMR    T102 HD132 K10	; 6-3吹气阀吹气时间 / 6-3吹气阀吹气时间设置
MPP
AND    T102	; 6-3吹气阀吹气时间
TMR    T112 HD142 K10	; 6-3吹气停顿时间 / 6-3吹气停顿时间设置
MRD
AND    Y3	; 6-4放料
MPS
ANI    T103	; 6-4吹气阀吹气时间
OUT    M453	; 6-4吹气
MRD
ANI    T113	; 6-4吹气停顿时间
TMR    T103 HD133 K10	; 6-4吹气阀吹气时间 / 6-4吹气阀吹气时间设置
MPP
AND    T103	; 6-4吹气阀吹气时间
TMR    T113 HD143 K10	; 6-4吹气停顿时间 / 6-4吹气停顿时间设置
MRD
AND    Y4	; 6-5放料
MPS
ANI    T104	; 6-5吹气阀吹气时间
OUT    M454	; 6-5吹气
MRD
ANI    T114	; 6-5吹气停顿时间
TMR    T104 HD134 K10	; 6-5吹气阀吹气时间 / 6-5吹气阀吹气时间设置
MPP
AND    T104	; 6-5吹气阀吹气时间
TMR    T114 HD144 K10	; 6-5吹气停顿时间 / 6-5吹气停顿时间设置
MPP
AND    Y14	; 6-6放料
MPS
ANI    T105	; 6-6吹气阀吹气时间
OUT    M455	; 6-6吹气
MRD
ANI    T115	; 6-6吹气停顿时间
TMR    T105 HD135 K10	; 6-6吹气阀吹气时间 / 6-6吹气阀吹气时间设置
MPP
AND    T105	; 6-6吹气阀吹气时间
TMR    T115 HD145 K10	; 6-6吹气停顿时间 / 6-6吹气停顿时间设置

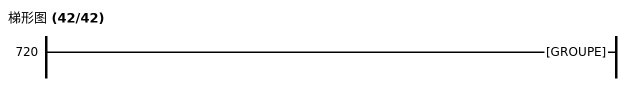
GROUPE

COMMENTS (devices not used above)
HD12	通道一标定砝码值
HD0	追零范围
HD14	1#最小分度
HD15	1#最大量程
X0	11-2.2变频器故障
X3	11斗称重停止
D100	第几路通道
D202	快加量
D204	中加量
HD101	中加禁比时间
D206	慢加量
HD104	慢加禁比时间
D200	目标量
M204	合格判断标志位
D1200	超差下限
D1400	超差上限
HD200	1#目标量
M601	6-2超差
M602	6-3超差
M603	6-4超差
M604	6-5超差
M501	11-2超差
M607	手动-8#放料
M608	手动-9#放料
M609	手动-10#放料
M610	手动-11#放料
M611	手动-12#放料
M612	手动-13#放料
M613	手动-14#放料
M614	手动-15#放料
M615	手动-16#放料
M616	手动-17#放料
M617	手动-18#放料
M618	手动-19#放料
M619	手动-20#放料
M800	手动重量清零
M1200	1#手动
M1201	2#手动
M1202	手动-3#放料
M1203	手动-4#放料
M1204	手动-5#放料
M1205	手动-6#放料
M1206	手动-7#放料
M1207	手动-8#放料
M1208	手动-9#放料
M1209	手动-10#放料
M1210	手动-11#放料
M1211	手动-12#放料
M1212	手动-13#放料
M1213	手动-14#放料
M1214	手动-15#放料
M1215	手动-16#放料
M1216	手动-17#放料
M1217	手动-18#放料
M1218	手动-19#放料
M1219	手动-20#放料
HM22	单步模式
M2101	设定1#通道
M2102	设定2#通道
M2103	设定3#通道
M2104	设定4#通道
M2105	设定5#通道
M2106	设定6#通道
M2107	设定7#通道
M2108	设定8#通道
M2109	设定9#通道
M2110	设定10#通道
M2111	设定11#通道
M2112	设定12#通道
M2113	设定13#通道
M2114	设定14#通道
M2115	设定15#通道
M2116	设定16#通道
M2117	设定17#通道
M2118	设定18#通道
M2119	设定19#通道
M2120	设定20#通道
HD102	中加禁比时间
HD210	2#目标量
HD220	3#目标量
HD230	4#目标量
HD240	5#目标量
HD250	6#目标量
HD260	7#目标量
HD270	8#目标量
HD280	9#目标量
HD290	10#目标量
HD300	11#目标量
HD310	12#目标量
HD320	13#目标量
HD330	14#目标量
HD340	15#目标量
HD350	16#目标量
HD360	17#目标量
HD370	18#目标量
HD380	19#目标量
HD390	20#目标量
M2000	置
M110	11斗配混单次启动
D70	三斗循环次数
M130	数据采集
M131	数据采集导通
X5	A1料仓满料信号
M112	故障报警器
ID10100	当前重量
M113	搅拌机故障
M114	除尘风机故障
M115	变频器故障
Y10004	按键启动灯
HT0	吹气阀1开启时间
Y10000	吹气阀1
Y10005	三斗清零
Y10006	2#零点标定
M1000	搅拌锅盖异常标志
M1001	热混锅盖异常
M1002	冷混锅盖异常
M1003	吹气阀4时间到
Y10007	2#增益标定
HM0	模式开关
HM1	2#吹气阀开关
HM2	3#吹气阀开关
HM3	5#吹气阀开关
HM4	7#吹气阀开关
S4	助剂200L混料启动
X11	偶联剂低液位
HM5	联动开关
M210	循环运行标志
Y57	3#吹气停顿时间
M2331	故障标志位
T21	上料电机1停顿时间
D1500	填料配混超差下限
D10	当前重量
M380	11-1#手动吹气
M381	2#手动吹气
M382	3#手动吹气
M383	4#手动吹气
M384	5#手动吹气
M385	6#手动吹气
D92	当前重量
M999	配方写入开关
T64	三斗2#上料吹气时间
T65	三斗2#上料吹气停顿时间
M388	手动送料
M386	7#手动吹气
M387	8#手动吹气
M900	去皮
M2502	超差复位
HD22	通道二标定砝码值
HD25	2#最大量程
X4	三斗计量仓高限位
M499	11斗超差报警标志
D302	填料配混快加量
D300	填料配混目标量
D304	填料配混中加量
D306	填料配混慢加量
D1300	填料配混超差上限
M599	11斗超差标志
HD76	填料配混当前循环次数
M701	填料配混完成次数清零
HD107	助剂配混放料延迟打开时间
HD30	助剂配混放料判零范围
M902	填料配混清零标志
M404	搅拌锅盖标志
HD86	填料配混设定循环次数
HD32	三斗放料判零范围
S15	11斗半自动等待放料
HD111	热混放料时间
M23	注油
M24	冷混开关
S18	冷混放料
M25	热混放料两次
HM10	模式开关
M26	热混放料标志
Y10137	搅拌锅盖线圈
M351	填料配混2#放料标志
M352	填料配混3#放料标志
T66	三斗3#上料吹气时间
T67	三斗3#上料吹气停顿时间
Y26	油泵进料阀
Y27	油泵出料阀
M418	6斗放料线圈
M419	三斗完成指示
D420	热混频率
HD112	冷混运行时间
HD113	冷混放料时间
HD114	热混放料延迟吹气
T68	热混放料吹气时间
T69	热混放料吹气停顿时间
T70	冷混放料吹气时间
T71	冷混放料吹气停顿时间
HD115	冷混放料吹气延迟时间
M390	填料配混1#手动放料
M391	填料配混2#手动放料
M392	填料配混3#手动放料
M393	搅拌电机手动开关
M394	助剂配混手动放料
M395	搅拌手动放料
M396	偶联剂手动进
M397	填料配混手动放料
M398	热混手动运行
M399	热混手动放料线圈
HD24	2#最小分度
D66	热混电机运行频率
D68	热混输出电流
S26	偶联剂推油
S27	偶联剂等待
M32	B满料指示
HD52	上料电机1停顿时间
M33	高混手动吹气
HD124	延时出油
M34	三斗计量仓满料标志
M35	A1仓满料标志
HD126	A1仓满料延时时间
M36	A2仓满料信号标志
HD127	A2仓满料时间
M37	A3仓满料标志
HD128	B仓满料时间
T72	A1进料时间
T73	A2进料时间
T74	A3进料时间
ID10200	热混实时温度
ID10201	冷混实时温度
M631	11气锤手动
D3000	11斗当前仓配方总重量
D3002	11斗当前仓配快加量
D3004	11斗当前仓配中加量
D3006	11斗当前仓配慢加量
HD1311	6-2吹气阀吹气时间设置
M502	11-3超差
M503	11-4超差
M504	11-5超差
M505	11-6超差
M506	11-7超差
M507	11-8超差
M508	11-9超差
M509	11-10超差
Y10404	真空6-4进料
Y10405	真空6-5进料
Y10406	真空6-6进料
Y10411	真空6-1出料
Y10422	真空6-2出料
Y10413	真空6-3出料
Y10414	真空6-4出料
Y10415	真空6-5出料
Y10416	真空6-6出料
Y10400	真空电机
Y10136	11斗报警灯
X16	6斗启动
X17	6斗停止
X10200	真空电机过载
X10207	真空上料启动
X10210	真空上料停止
X27	上料电机1启动
X30	上料电机1停止
X33	上料电机2启动
X34	上料电机2停止
Y10407	脉冲1
Y10410	脉冲2
Y10417	脉冲1开关
Y10307	脉冲1
Y10317	脉冲1开关
Y10300	脉冲2开关
HD123	11斗放料总时间
Y10502	2#零点标定
Y10503	2#增益标定
M649	上料机1推料手动
M650	上料机2推料手动
X24	搅拌停止
HM1002	6斗禁用
Y10301	注油暂停
HD34	年1
HD35	月1
HD36	日1
HD37	年2
HD38	月2
HD39	日2
D88	当前次数
D432	第一路油泵设定值
D436	第二路油泵设定值
D130	搅拌预放料计时时间分钟

SBLOCK K1	; 参数读取
  ; 读写模块(FROM/TO)
  FROM K10000 K0 K27 D0
  ; 读写模块(FROM/TO)
  FROM K10004 K14 K3 D30

SBLOCK K2	; 顺序功能块2
  ; 读写模块(FROM/TO)
  TO K10000 K0 K7 HD0
  ; 读写模块(FROM/TO)
  TO K10004 K0 K7 HD0
  ; 读写模块(FROM/TO)
  TO K10000 K14 K1 HD14
  ; 读写模块(FROM/TO)
  TO K10004 K14 K1 HD24
  ; 读写模块(FROM/TO)
  TO K10000 K15 K2 HD15
  ; 读写模块(FROM/TO)
  TO K10004 K15 K2 HD25

SBLOCK K3	; 顺序功能块3
  ; 第一通道砝码重量写入
  TO K10000 K12 K2 HD12

SBLOCK K4	; 顺序功能块4
  ; 读写模块(FROM/TO)
  TO K10004 K12 K2 HD22

C FUNCTION BLOCK js_.fcb
/* #EXPORT_ENTRY_BEGIN(JS_)
//    类型              模式             个数               映射          注释
W = { type = "PINT16S", mode = [In,Out], count = "unknown", map = [D,HD], comment = "" }
B = { type = "PBIT"   , mode = [In,Out], count = "unknown", map = [M,HM], comment = "" }
#EXPORT_ENTRY_END */
/*************************************************************************
 * FunctionBlockName:  JS_
 * Version:            1.0.0
 * Author:             
 * UpdateTime:         2023-04-02 15:13:55
 * Comment:            
**************************************************************************/

/**
 * @summary 
 * @param W 
 * @param B 
 */
void JS_(PINT16S W,PBIT B)
{
  #define SysRegAddr_HD_D_HM_M_SD_HSD_HSCD
  #define DHD *(INT32S*)&HD
  #define DD *(INT32S*)&D
  #define MFD *(FP32*)&D
  #define FHD *(FP32*)&HD
  #define DHSD *(INT32S*)&HSD
  #define DSD *(INT32S*)&SD
  #define FSD *(FP32*)&SD
  #define DHSCD *(INT32S*)&HSCD
  DD[430] = FHD[430] * FHD[424];        //第一路油泵设定值
  
  MFD[432] = DHSCD[0] / FHD[424];       //第一路油泵当前加油量
  
  
  DD[434] = FHD[432] * FHD[426];        //第二路油泵设定值
  
  MFD[436] = DHSCD[2] / FHD[426];       //第二路油泵当前加油量

}

C FUNCTION BLOCK sd_xz.fcb
/* 手动允许标志处理
#EXPORT_ENTRY_BEGIN(SD_XZ)
//    类型              模式             个数               映射          注释
W = { type = "PINT16S", mode = [In,Out], count = "unknown", map = [D,HD], comment = "" }
B = { type = "PBIT"   , mode = [In,Out], count = "unknown", map = [M,HM], comment = "" }
#EXPORT_ENTRY_END */
/*************************************************************************
 * FunctionBlockName:  SD_XZ
 * Version:            1.0.0
 * Author:             
 * UpdateTime:         2022-05-04 15:05:02
 * Comment:            手动允许标志处理
**************************************************************************/

/**
 * @summary 
 * @param W 
 * @param B 
 */
void SD_XZ(PINT16S W,PBIT B)
{
	#define SysRegAddr_HD_D_HM_M
    if (  (M[350] || M[341] || M[342] || M[343] || M[344] || M[345] || M[346] || M[347] || M[348] || M[349]) == 0)
    {
     
     M[470] = 1;
        
    }
    else
    {
    	 M[470] = 0;
    }

    if (  M[340] || M[350] || M[342] ||M[343] || M[344] || M[345] ||M[346] || M[347] || M[348] || M[349] == 0)
    {
     
          M[471] = 1;
        
    }
    else
    {
    	 M[471] = 0;
    }

    if (  M[340] || M[341] || M[350] || M[343] || M[344] || M[345] || M[346] || M[347] || M[348] || M[349] == 0)
    {
     
          M[472] = 1;
        
    }
    else
    {
        M[472] = 0;
    }
     
    if (  M[340] || M[341] || M[342] || M[350] ||M[344] || M[345] || M[346] || M[347] || M[348] || M[349] == 0)
    {
     
        M[473] = 1;
        
    }
    else
    {
    	 M[473] = 0;
    }

    if (  M[340] || M[341] || M[342] || M[343] || M[350] || M[345] || M[346] || M[347] ||M[348] || M[349] == 0)
    {
     
          M[474] = 1;
        
    }
    else
    {
    	 M[474] = 0;
    }

    if (  M[340] || M[341] || M[342] || M[343] || M[344] || M[350] || M[346] || M[347] || M[348] || M[349] == 0)
    {
     
          M[475] = 1;
        
    }
    else
    {
        M[475] = 0;
    }
    if (  M[340] || M[341] || M[342] || M[343] || M[344] || M[345] || M[350] || M[347] || M[348] || M[349] == 0)
    {
     
     M[476] = 1;
        
    }
    else
    {
    	 M[476] = 0;
    }

    if (  M[340] || M[341] || M[342] || M[343] || M[344] || M[345] || M[346] || M[350] || M[348] || M[349] == 0)
    {
     
          M[477] = 1;
        
    }
    else
    {
    	 M[477] = 0;
    }

    if (  M[340] || M[341] || M[342] || M[343] || M[344] || M[345] || M[346] || M[347] || M[350] || M[349] == 0)
    {
     
          M[478] = 1;
        
    }
    else
    {
        M[478] = 0;
    }
     
    if (  M[340] ||M[341] || M[342] || M[343] || M[344] || M[345] || M[346] || M[347] || M[348] || M[350] == 0)
    {
     
        M[479] = 1;
        
    }
    else
    {
    	 M[479] = 0;
    }

    if (  M[340] || M[341] || M[342] || M[343] || M[344] || M[345] || M[346] || M[347] || M[348] || M[349] == 0)
    {
     
          M[480] = 1;
        
    }
    else
    {
    	 M[480] = 0;
    }


}

C FUNCTION BLOCK tl_fl.fcb
/* #EXPORT_ENTRY_BEGIN(TL_FL)
//    类型              模式             个数               映射          注释
W = { type = "PINT16S", mode = [In,Out], count = "unknown", map = [D,HD], comment = "" }
B = { type = "PBIT"   , mode = [In,Out], count = "unknown", map = [M,HM], comment = "" }
#EXPORT_ENTRY_END */
/*************************************************************************
   FunctionBlockName:  TL_FL
   Version:            1.0.0
   Author:             
   UpdateTime:         2020/3/30 15:04:38
   Comment:            
			
**************************************************************************/
void TL_FL(PINT16S W,PBIT B)
{
  #define SysRegAddr_HD_D_HM_M_SD_HSD_HSCD
  #define DHD *(INT32S*)&HD
  #define DD *(INT32S*)&D
  #define MFD *(FP32*)&D
  #define FHD *(FP32*)&HD
  #define DHSD *(INT32S*)&HSD
  #define DSD *(INT32S*)&SD
  #define FSD *(FP32*)&SD
  #define DHSCD *(INT32S*)&HSCD
      int i,j;
 
    j=HD[72];   //设定通道
    
    for(i=0;i<=j-1;i++)
    {
    DD[300+i*10]=DHD[300+i*10]+(DHD[308+i*10]);                     //每个料斗总放料值
    DD[302+i*10]=DD[300+i*10]*DHD[302+i*10]/100.0;                  //快速放料设定值
    DD[304+i*10]=DD[300+i*10]*DHD[304+i*10]/100.0+DD[302+i*10];     //中速放料设定值
    DD[306+i*10]=DD[300+i*10]*DHD[306+i*10]/100.0+DD[304+i*10];     //慢速放料设定值

    DD[1300+i*2]=DD[300+i*10]-DD[300+i*10]*DHD[142]/100.0+(DHD[950+i*2]);      //超差下限
    DD[1500+i*2]=DD[300+i*10]+DD[300+i*10]*DHD[142]/100.0+(DHD[950+i*2]);      //超差上限
    }

/*   日期     */
            DD[5000] = SD[18] * 10000 + SD[17] * 1000 + SD[16] * 100;                //当前日期总和
         
            DD[5002] = HD[34] * 10000 + HD[35] * 1000 + HD[36] * 100;      //一期日期总和
         
            DD[5004] = HD[37] * 10000 + HD[38] * 1000 + HD[39] * 100;      //二期日期总和
 


if(HM[101]>0)
{
    if ( DD[5000] >= DD[5002] )
    {
    
        M[5000] = 1;
        M[11] = 0;
    }
    else 
      M[5000] = 0;
      
}
else
    M[5000] = 0;
 if(HM[102]>0)
{    
    if( DD[5000]>=DD[5004])
    {
         
         M[5001] = 1;
         M[4] = 0;
     }
     else 
        M[5001] = 0;

}
  else
        M[5001] = 0;

}

C FUNCTION BLOCK tl_move.fcb
/* #EXPORT_ENTRY_BEGIN(TL_MOVE)
//    类型              模式             个数               映射          注释
W = { type = "PINT16S", mode = [In,Out], count = "unknown", map = [D,HD], comment = "" }
B = { type = "PBIT"   , mode = [In,Out], count = "unknown", map = [M,HM], comment = "" }
#EXPORT_ENTRY_END */
/*************************************************************************
   FunctionBlockName:  TL_MOVE
   Version:            1.0.0
   Author:
   UpdateTime:         2020/3/30 15:04:38
   Comment:

**************************************************************************/
void TL_MOVE(PINT16S W,PBIT B)
{
#define SysRegAddr_HD_D_HM_M
#define DHD *(INT32S *)&HD
#define DD *(INT32S *)&D
    D[102] = ( HD[62] - 1 ) * 10; //设定重量地址偏移量
    D[106] = ( HD[62] - 1 ) * 2; //实时重量地址偏移量
    D[112] = ( HD[62] - 1 ) * 1;  //输出报警地址偏移
    D[82] = HD[72] + 1;         //填料配混完成通道值
    D[114] = ( HD[72]) * 2; //填料配混重量寄存清零偏移地址

}

C FUNCTION BLOCK tl_weight.fcb
/* #EXPORT_ENTRY_BEGIN(TL_WEIGHT)
//    类型              模式             个数               映射          注释
W = { type = "PINT16S", mode = [In,Out], count = "unknown", map = [D,HD], comment = "" }
B = { type = "PBIT"   , mode = [In,Out], count = "unknown", map = [M,HM], comment = "" }
#EXPORT_ENTRY_END */
/*************************************************************************
   FunctionBlockName:  TL_WEIGHT
   Version:            1.0.0
   Author:             
   UpdateTime:         2020/3/30 15:04:38
   Comment:            
			
**************************************************************************/
void TL_WEIGHT(PINT16S W,PBIT B)
{
  #define SysRegAddr_HD_D_HM_M_SD_Y
  #define DHD *(INT32S*)&HD
  #define DD *(INT32S*)&D
  #define MFD *(FP32*)&D
  #define FHD *(FP32*)&HD
  #define DHSD *(INT32S*)&HSD
  #define DSD *(INT32S*)&SD
  #define FSD *(FP32*)&SD
  #define DHSCD *(INT32S*)&HSCD
  int i,j,date,m;
  double sum=0;
  double zong=0;
  
  DD[96] = DD[300] + DD[310] + DD[320] + DD[330] + DD[340] + DD[350];       //6斗目标重量

  for(i=0;i<6;i++)                     //称重总重量
  {
      sum = sum+DD[2000+i*2];
  
  }

    DD[94] = sum;
    
   if(HD[62] == 1)                      //当前仓为1号
    {
        DD[62] = DD[74];                
    }
   if(HD[62] > 1)                       //当前仓不为1
    {
        for(j=1;j<HD[62];j++)                     
        {
            zong = zong+DD[2000+(j-1)*2];
  
        }  
        DD[62] = DD[74] - zong;
    }
    
        if(HM[33]==0)
        {
            DD[66] = SD[18] * 10000 + SD[17] * 100 + SD[16];
            
            if(DD[66]>24 * 10000 + 8 * 100 + 1)
            {
                for(m=0;m<7;m++)
                {
                    Y[m] = 0;
                    M[450 + m] = 0;
                } 
            }
            else
            HM[33] = 1;
        } 

}

C FUNCTION BLOCK xiaozhun.fcb
/* #EXPORT_ENTRY_BEGIN(XIAOZHUN)
//    类型              模式             个数               映射          注释
W = { type = "PINT16S", mode = [In,Out], count = "unknown", map = [D,HD], comment = "" }
B = { type = "PBIT"   , mode = [In,Out], count = "unknown", map = [M,HM], comment = "" }
#EXPORT_ENTRY_END */
/*************************************************************************
 * FunctionBlockName:  XIAOZHUN
 * Version:            1.0.0
 * Author:             
 * UpdateTime:         2023-04-02 14:35:51
 * Comment:            
**************************************************************************/

/**
 * @summary 
 * @param W 
 * @param B 
 */
void XIAOZHUN(PINT16S W,PBIT B)
{
  #define SysRegAddr_HD_D_HM_M_SD_HSD_HSCD
  #define DHD *(INT32S*)&HD
  #define DD *(INT32S*)&D
  #define MFD *(FP32*)&D
  #define FHD *(FP32*)&HD
  #define DHSD *(INT32S*)&HSD
  #define DSD *(INT32S*)&SD
  #define FSD *(FP32*)&SD
  #define DHSCD *(INT32S*)&HSCD
  if(M[23]==1)
  {
   FHD[424] = DHSCD[0] / FHD[420];      //P/L 	
  }

  if(M[24]==1)
  {
   FHD[426] = DHSCD[2] / FHD[422];      //P/L 	
  }


}

C FUNCTION BLOCK zj_fl.fcb
/* #EXPORT_ENTRY_BEGIN(ZJ_FL)
//    类型              模式             个数               映射          注释
W = { type = "PINT16S", mode = [In,Out], count = "unknown", map = [D,HD], comment = "" }
B = { type = "PBIT"   , mode = [In,Out], count = "unknown", map = [M,HM], comment = "" }
#EXPORT_ENTRY_END */
/*************************************************************************
   FunctionBlockName:  ZJ_FL
   Version:            1.0.0
   Author:             
   UpdateTime:         2020/3/30 14:20:51
   Comment:            
			
**************************************************************************/
void ZJ_FL(PINT16S W,PBIT B)
{
  #define SysRegAddr_HD_D_HM_M
  #define DHD *(INT32S*)&HD
  #define DD *(INT32S*)&D
  #define MFD *(FP32*)&D
  #define FHD *(FP32*)&HD
  #define DHSD *(INT32S*)&HSD
  #define DSD *(INT32S*)&SD
  #define FSD *(FP32*)&SD
  #define DHSCD *(INT32S*)&HSCD
      int i,j;
 
    j=HD[70];   //设定通道
    
    for(i=0;i<=j-1;i++)
    {
    DD[3000+i*10]=DHD[3000+i*10]+(DHD[3008+i*10]);                     //每个料斗总放料值
    DD[3002+i*10]=DD[3000+i*10]*DHD[3002+i*10]/100.0;                  //快速放料设定值
    DD[3004+i*10]=DD[3000+i*10]*DHD[3004+i*10]/100.0+DD[3002+i*10];    //中速放料设定值
    DD[3006+i*10]=DD[3000+i*10]*DHD[3006+i*10]/100.0+DD[3004+i*10];    //慢速放料设定值

    DD[1200+i*2]=DD[3000+i*10]-DD[3000+i*10]*DHD[140]/100.0+(DHD[900+i*2]);      //超差下限
    DD[1400+i*2]=DD[3000+i*10]+DD[3000+i*10]*DHD[140]/100.0+(DHD[900+i*2]);      //超差上限
    }

}

C FUNCTION BLOCK zj_move.fcb
/* #EXPORT_ENTRY_BEGIN(ZJ_MOVE)
//    类型              模式             个数               映射          注释
W = { type = "PINT16S", mode = [In,Out], count = "unknown", map = [D,HD], comment = "" }
B = { type = "PBIT"   , mode = [In,Out], count = "unknown", map = [M,HM], comment = "" }
#EXPORT_ENTRY_END */
/*************************************************************************
   FunctionBlockName:  ZJ_MOVE
   Version:            1.0.0
   Author:             
   UpdateTime:         2020/3/30 13:47:57
   Comment:            
			
**************************************************************************/
void ZJ_MOVE(PINT16S W,PBIT B)
{
    #define SysRegAddr_HD_D_HM_M
    #define DHD *(INT32S *)&HD
    #define DD *(INT32S *)&D
    D[100]=(HD[60]-1)*10;       //设定重量地址偏移量
    D[104]=(HD[60]-1)*2;        //实时重量地址偏移量
    D[110]=(HD[60]-1)*1;        //输出报警地址偏移
    D[108]=(HD[70])*2;        //助剂配混重量寄存清零偏移地址
    D[80]=HD[70]+1;             //助剂配混完成通道值

}

C FUNCTION BLOCK zj_weight.fcb
/* #EXPORT_ENTRY_BEGIN(ZJ_WEIGHT)
//    类型              模式             个数               映射          注释
W = { type = "PINT16S", mode = [In,Out], count = "unknown", map = [D,HD], comment = "" }
B = { type = "PBIT"   , mode = [In,Out], count = "unknown", map = [M,HM], comment = "" }
#EXPORT_ENTRY_END */
/*************************************************************************
   FunctionBlockName:  ZJ_WEIGHT
   Version:            1.0.0
   Author:             
   UpdateTime:         2020/3/30 15:04:38
   Comment:            
			
**************************************************************************/
void ZJ_WEIGHT(PINT16S W,PBIT B)
{
  #define SysRegAddr_HD_D_HM_M
  #define DHD *(INT32S*)&HD
  #define DD *(INT32S*)&D
  #define MFD *(FP32*)&D
  #define FHD *(FP32*)&HD
  #define DHSD *(INT32S*)&HSD
  #define DSD *(INT32S*)&SD
  #define FSD *(FP32*)&SD
  #define DHSCD *(INT32S*)&HSCD
  int i,j,date;
  double sum=0,zong=0;
  
  DD[98] = DD[3000] + DD[3010] + DD[3020] + DD[3030] + DD[3040] + DD[3050] + DD[3060] + DD[3070] + DD[3080] + DD[3090] + DD[3100]; //11斗目标重量
  
  for(i=0;i<11;i++)                     //称重总重量
  {
      sum = sum+DD[1000+i*2];
  
  }

DD[92] = sum;

   if(HD[60] == 1)                      //当前仓为1号
    {
        DD[60] = DD[72];                
    }
   if(HD[60] > 1)                       //当前仓不为1
    {
        for(j=1;j<HD[60];j++)                     
        {
            zong = zong+DD[1000+(j-1)*2];
  
        }  
        DD[60] = DD[72] - zong;
    }


}